// TwinCAT 3 PLC project PLC_1
// ProgramVersion: 3.1.4024.0
// libraries:
//   Tc2_Standard, * (Beckhoff Automation GmbH)
//   Tc2_System, * (Beckhoff Automation GmbH)
//   Tc3_Module, * (Beckhoff Automation GmbH)
// project tree:
//   GVLs/ HMI.TcGVL
//   / PlcTask.TcTTO
//   POUs/ FB_Array.TcPOU, FB_Check.TcPOU, MAIN.TcPOU

CONFIGURATION PLC_1
    RESOURCE PLC ON TwinCAT3
        TASK PlcTask(INTERVAL := T#10ms, PRIORITY := 20);
        PROGRAM MAIN WITH PlcTask : MAIN;
    END_RESOURCE
END_CONFIGURATION

// ---- GVLs/HMI.TcGVL
{attribute 'qualified_only'}
VAR_GLOBAL
	iPageNumber :INT:=1;
	xButton1:BOOL;
	xButton2:BOOL;
	xButton3:BOOL;
	xButton4:BOOL;
	xButton5:BOOL;
	xButton6:BOOL;
END_VAR

// ---- POUs/MAIN.TcPOU
PROGRAM MAIN
VAR
	fb_array:FB_Array;
	fb_check:FB_Check;
END_VAR

fb_array();
fb_check();
// Setting value to iPageNumber when button is pressed
IF HMI.xButton1 THEN
	HMI.iPageNumber:=1;
	HMI.xButton1:=FALSE;
ELSIF HMI.xButton2 THEN
	HMI.iPageNumber:=2;
	HMI.xButton2:=FALSE;
ELSIF HMI.xButton3 THEN
	HMI.iPageNumber:=3;
	HMI.xButton3:=FALSE;
ELSIF HMI.xButton4 THEN
	HMI.iPageNumber:=4;
	HMI.xButton4:=FALSE;
ELSIF HMI.xButton5 THEN
	HMI.iPageNumber:=5;
	HMI.xButton5:=FALSE;
ELSIF HMI.xButton6 THEN
	HMI.iPageNumber:=6;	
	HMI.xButton6:=FALSE;					
END_IF

END_PROGRAM

// ---- POUs/FB_Array.TcPOU
FUNCTION_BLOCK FB_Array
VAR_INPUT
END_VAR
VAR_OUTPUT
	
END_VAR
VAR
	aArray : ARRAY[0..19] OF LREAL;  // Creating array with 20 cells
	dDRAND : DRAND;                  // Random number generator
	xCycle :BOOL:=TRUE;              // Variable ending program after one cycle
	iCellNumber:INT; 
    aTestArray2    : ARRAY[0..19] OF LREAL;
    udiMoveResult : UDINT; 
	xMoveArrayElements:BOOL:=FALSE;       
END_VAR

dDRAND(Seed:= , Num=> );               // Generating random number
IF xCycle THEN                  	   
    FOR iCellNumber := 0 TO 19 DO	   // Setting numbers of cells in array to 20
        dDRAND();                
        aArray[iCellNumber] := dDRAND.Num;  // Creating array
    END_FOR;
    xCycle := FALSE;                        // Ending cycle
END_IF
// Moving elements in array down if bool variable is TRUE
IF xMoveArrayElements THEN
	MEMMOVE(ADR(aArray[1]), ADR(aArray[0]), SIZEOF(aArray) - SIZEOF(aArray[0]));	// Writing value from previous cell to another and deleting the last one
 	xMoveArrayElements:=FALSE;			// Ending loop
	aArray[0] := 1.0; 					// Setting value one to first cell
END_IF

//udiMoveResult := MEMMOVE(ADR(aTestArray2), ADR(aArray), SIZEOF(aArray));   // Moving numbers from first array one down to another array
//aTestArray2[0]:=1;														// Setting 0 in 1st cell in array,

END_FUNCTION_BLOCK

// ---- POUs/FB_Check.TcPOU
FUNCTION_BLOCK FB_Check
VAR_INPUT
END_VAR
VAR_OUTPUT
END_VAR
VAR
	axTest: ARRAY[0..19] OF BOOL;    // Array of 20 Bool type elements
	iCell: INT;						 
	x:BOOL:=TRUE;
	iNumberOfCellWithTrueValue:INT;					// Number of cell where bool value is true
	xEndingLoop: BOOL:=FALSE;				// Variable ending loop when there is true value in array
END_VAR

// Method 
CheckIfAnyArrayElementsTrue();
// Setting values to array
IF 	NOT xEndingLoop THEN
	FOR iCell:= 0 TO 19 DO	
		// True value in 7th cell
		IF iCell = 7  THEN
			axTest[iCell]:=TRUE;
			xEndingLoop:=TRUE;
		ELSE
			axTest[iCell]:=FALSE;
		
		END_IF
	END_FOR
	xEndingLoop:=TRUE;
ELSE
	;
END_IF

METHOD CheckIfAnyArrayElementsTrue : BOOL
VAR_INPUT
END_VAR
VAR_INST
	xInArrayExistsTrueValue:BOOL;
END_VAR
// Loop ending when xCell = TRUE
IF x:=TRUE THEN
	FOR iCell:= 0 TO 19  DO
		// Searching TRUE value in array
		IF axTest[iCell]= TRUE THEN
			iNumberOfCellWithTrueValue:=iCell;
			x:=FALSE;
			xInArrayExistsTrueValue:=TRUE;
			EXIT;
		END_IF
	END_FOR
END_IF
END_METHOD

END_FUNCTION_BLOCK
